FUNCTION_BLOCK NamespaceExtractor
VAR_OUTPUT
	{attribute 'init_namespace'} 
	CurrentNamespace : STRING(255);	
END_VAR

END_FUNCTION_BLOCK

(* stored: Version 1.1.0.1
   POU NamespaceExtractor: Id {ec23540e-4f6e-4415-bd00-943358bc77a2}, SpecialFunc None *)
